// TwinCAT 3 PLC project Proj_Ueb_sw01
// ProgramVersion: 3.1.4023.0
// libraries:
//   Tc2_Standard, * (Beckhoff Automation GmbH)
//   Tc2_System, * (Beckhoff Automation GmbH)
//   Tc3_Module, * (Beckhoff Automation GmbH)
// project tree:
//   DUTs/ En_DistanceMode.TcDUT, En_ToggleMode.TcDUT
//   GVLs/ GVL_IO.TcGVL
//   / PlcTask.TcTTO
//   POUs/ Fb_MeanCalculatorWForgettingFactor.TcPOU, Fb_EdgeDetector.TcPOU, Fb_UltrasonicSensor.TcPOU, FUN_0to10V_TO_INT.TcPOU, FUN_Add.TcPOU, FUN_Divide.TcPOU, FUN_Multiply.TcPOU, FUN_Substract.TcPOU, MAIN.TcPOU, FUN_ShiftLeft.TcPOU, FUN_MeanCalculator.TcPOU, PRG_DoSomeMath.TcPOU
// (motion and I/O tree: see PLC project proj_sw01)
// real-time tasks:
//   TASK PlcTask: cycle T#10ms, priority 20, ADS port 350
//   TASK PlcTask1: cycle T#10ms, priority 21, ADS port 351
//   TASK PlcTask2: cycle T#10ms, priority 22, ADS port 352
// variable links:
//   Proj_Ueb_sw01/Proj_Ueb_sw01 Instance <-> Device 1 (EtherCAT)/Term 1 (EK1200)/Term 2 (EL1004)
//     PlcTask Inputs/GVL_IO.DI_BtnBlue <-> Channel 2/Input
//     PlcTask Inputs/GVL_IO.DI_BtnYellow <-> Channel 1/Input
//   Proj_Ueb_sw01/Proj_Ueb_sw01 Instance <-> Device 1 (EtherCAT)/Term 1 (EK1200)/Term 3 (EL2004)
//     PlcTask Outputs/GVL_IO.DO_LampGreen <-> Channel 2/Output
//     PlcTask Outputs/GVL_IO.DO_LampRed <-> Channel 1/Output
//   Proj_Ueb_sw01/Proj_Ueb_sw01 Instance <-> Device 1 (EtherCAT)/Term 1 (EK1200)/Term 4 (EL3004)
//     PlcTask Inputs/GVL_IO.AI_UltraSonicSensor <-> AI Standard Channel 1/Value
//   Proj_Ueb_sw01/Proj_Ueb_sw01 Instance <-> Device 1 (EtherCAT)/Term 1 (EK1200)/Term 5 (EL4034)
//     PlcTask Outputs/GVL_IO.AO_AnalogGauge <-> AO Outputs Channel 1/Analog output

CONFIGURATION Proj_Ueb_sw01
    RESOURCE PLC ON TwinCAT3
        TASK PlcTask(INTERVAL := T#10ms, PRIORITY := 21);
        PROGRAM MAIN WITH PlcTask : MAIN;
    END_RESOURCE
END_CONFIGURATION

// ---- DUTs/En_DistanceMode.TcDUT
{attribute 'qualified_only'}
{attribute 'strict'}
TYPE En_DistanceMode :
(
	Default := 0,
	NearerIsHigher,
	NearerIsLower
);
END_TYPE

// ---- DUTs/En_ToggleMode.TcDUT
{attribute 'qualified_only'}
{attribute 'strict'}
TYPE En_ToggleMode :
(
	Off := 0,
	Simulataneous,
	Alternating
);
END_TYPE

// ---- GVLs/GVL_IO.TcGVL
{attribute 'qualified_only'}
VAR_GLOBAL
	DI_BtnYellow 	AT %I* : BOOL;
	DI_BtnBlue	 	AT %I* : BOOL;
	
	DO_LampRed 		AT %Q* : BOOL;
	DO_LampGreen	AT %Q* : BOOL;
	
	AI_UltraSonicSensor  AT %I* : INT;
	AO_AnalogGauge		 AT %Q* : INT;
END_VAR

// ---- POUs/MAIN.TcPOU
PROGRAM MAIN
VAR
	f_Result 			:	REAL;
	i_Counter			: 	INT;
	f_RandomArray		: 	ARRAY[1..10] OF REAL := [5.0, 3.5, 4.6, 1.2, 13, 5.4, 5.6, 11.0, 15.6, 10];
	f_Product			: 	REAL;
	f_Sum 				: 	REAL;
	
	edgeDetectorBtnY	:   Fb_EdgeDetector;
	edgeDetectorBtnB	:   Fb_EdgeDetector;
	t_ToggleTime		: 	TIME := T#333MS;	// 1/Hz = [s]
	t_lastToggle		: 	TIME := TIME();
	togglingMode		: 	En_ToggleMode := En_ToggleMode.Off;
	b_LampR_On			: 	BOOL := FALSE;
	b_LampG_On			: 	BOOL := FALSE;
	
	ultraSonicSensorFb	:	Fb_UltrasonicSensor;
	
	a_lastValues		: 	ARRAY [1..NUM_STORED_VALS] OF REAL; 
	r_meanVal			: 	REAL := 0;
	fb_MeanCalc			: 	Fb_MeanCalculatorWForgettingFactor;
	r_forgettingFactor	: 	REAL := 0.5;
END_VAR
VAR CONSTANT
	NUM_STORED_VALS		: INT := 300;
END_VAR

// Aufgabe 1
f_Result := FUN_Add(1.3, 1.5);
f_Result := FUN_Add(3.3, 1000.5);
f_Result := FUN_Add(5.5, 51.5);

f_Result := FUN_Substract(1.3, 1);
f_Result := FUN_Substract(1.3, 2);

f_Result := FUN_Multiply(3, 1000);
f_Result := FUN_Multiply(55, 5.55);

f_Result := FUN_Divide(9, 3);
f_Result := FUN_Divide(55, 0);


// Aufgabe 3
// Call program
PRG_DoSomeMath.f_Inp1 := 1.5;
PRG_DoSomeMath.f_Inp2 := 5.4;
PRG_DoSomeMath();
// Access program variables
f_Result := PRG_DoSomeMath.f_AddResult;
i_Counter := PRG_DoSomeMath.i_CallCounter;


// Aufgabe 7 & 8
// insert first values
f_Product := f_RandomArray[1];
f_Sum := f_RandomArray[1];
// for loop
FOR i_Counter := 2 TO 10 DO
	f_Product 	:= f_Product * f_RandomArray[i_Counter];
	f_Sum		:= f_Sum + f_RandomArray[i_Counter];
END_FOR

// Aufgabe 9
// insert first values
f_Product := f_RandomArray[1];
f_Sum := f_RandomArray[1];
i_Counter := 2;
// while loop
WHILE i_Counter <= 10 DO
	f_Product 	:= f_Product * f_RandomArray[i_Counter];
	f_Sum		:= f_Sum + f_RandomArray[i_Counter];
	i_Counter 	:= i_Counter + 1;
END_WHILE

// Aufgabe 10
// insert first values
f_Product := f_RandomArray[1];
f_Sum := f_RandomArray[1];
i_Counter := 2;
// do while loop = repeat loop
REPEAT
	f_Product 	:= f_Product * f_RandomArray[i_Counter];
	f_Sum		:= f_Sum + f_RandomArray[i_Counter];
	i_Counter 	:= i_Counter + 1;
UNTIL i_Counter > 10
END_REPEAT


// Aufgabe 11 and 12
edgeDetectorBtnY(inputValue := GVL_IO.DI_BtnYellow);
edgeDetectorBtnB(inputValue := GVL_IO.DI_BtnBlue);

// double press?
IF edgeDetectorBtnB.doublePress OR edgeDetectorBtnY.doublePress THEN
	t_ToggleTime := t_ToggleTime / 2;  // double frequency
END_IF

// triple press?
IF edgeDetectorBtnB.triplePress OR edgeDetectorBtnY.triplePress THEN
	t_ToggleTime := t_ToggleTime * 2;  // half frequency
END_IF

CASE togglingMode OF
	
	/// CASE OFF ///
	En_ToggleMode.Off:
	// lamp actions
	b_LampR_On := FALSE;
	b_LampG_On := FALSE;
	t_ToggleTime := T#333MS; // reset to default time
	
	// switch mode
	IF edgeDetectorBtnY.risingEdge THEN
		togglingMode := En_ToggleMode.Simulataneous;
	END_IF
	IF edgeDetectorBtnB.risingEdge THEN 
		togglingMode := En_ToggleMode.Alternating;
		b_LampG_On := TRUE;  // initial lamp on => alternating
	END_IF
	
	/// CASE Simulataneous ///
	En_ToggleMode.Simulataneous:
	// lamp actions
	IF((t_lastToggle + t_ToggleTime) < TIME()) THEN
		b_LampR_On := NOT b_LampR_On;
		b_LampG_On := NOT b_LampG_On;
		t_lastToggle := TIME();
	END_IF
	
	// switch mode
	IF edgeDetectorBtnY.risingEdge THEN
		togglingMode := En_ToggleMode.Off;
	END_IF
	

	/// CASE ALTERNATING ///
	En_ToggleMode.Alternating:
	// lamp actions
	IF((t_lastToggle + t_ToggleTime) < TIME()) THEN
		b_LampR_On := NOT b_LampR_On;
		b_LampG_On := NOT b_LampG_On;
		t_lastToggle := TIME();
	END_IF
	
	// switch mode
	IF edgeDetectorBtnB.risingEdge THEN
		togglingMode := En_ToggleMode.Off;
	END_IF

	
END_CASE


GVL_IO.DO_LampRed := b_LampR_On;
GVL_IO.DO_LampGreen := b_LampG_On;


// Aufgabe 13
ultraSonicSensorFb(	i_UltraSonicAnalogInput := GVL_IO.AI_UltraSonicSensor, 
					e_DistanceMode := En_DistanceMode.NearerIsHigher);
GVL_IO.AO_AnalogGauge := ultraSonicSensorFb.i_AnalogOutput;

// Aufgabe 14
FUN_ShiftLeft(a_Values := a_lastValues);  // shift array left
a_lastValues[NUM_STORED_VALS] := ultraSonicSensorFb.r_VoltageUltraSonicSensor;  // store last value

// Aufgabe 15
fb_MeanCalc(r_inputValue := ultraSonicSensorFb.r_VoltageUltraSonicSensor, r_forgettingFactor := r_forgettingFactor);
r_meanVal := fb_MeanCalc.r_meanValueOutput;
GVL_IO.AO_AnalogGauge := FUN_0to10V_TO_INT(r_AnalogValue0to10V := r_meanVal);

END_PROGRAM

// ---- POUs/Fb_EdgeDetector.TcPOU
FUNCTION_BLOCK INTERNAL Fb_EdgeDetector
VAR_INPUT
	inputValue		: BOOL;
END_VAR
VAR_OUTPUT
	risingEdge		: BOOL;
	fallingEdge		: BOOL;
	doublePress		: BOOL;
	triplePress		: BOOL;
END_VAR
VAR
	i_risingEdgCnt			: INT := 0;  		// internal var
	lastValue 				: BOOL;				// last value registered
	tlastPush				: TIME := TIME();	// time when last push happened
	tLastRising				: TIME := TIME();	// time when last rising edge happened
	tDebounce	    		: TIME := T#20MS;   // time to debounce input value
	tMultiPressTime			: TIME := T#200MS;	// time between which multiple presses to allow the user to press button again
	
END_VAR

// reset output signals
fallingEdge := FALSE;
risingEdge := FALSE;
doublePress := FALSE;
triplePress := FALSE;

// if a change happened and new values get accepted
IF(inputValue <> lastValue AND (tlastPush + tDebounce) < TIME()) THEN
	IF(inputValue) THEN
		i_risingEdgCnt := i_risingEdgCnt + 1;
		
		tLastRising := TIME(); // reset last rising time (give another tMultiPressTime time to press the button another time
	ELSE
		fallingEdge := TRUE;
	END_IF
	lastValue := inputValue;  // overwrite stored value
	tlastPush := TIME();
END_IF


// handle rising edge (with double press)
CASE i_risingEdgCnt OF
	1:
	IF (tLastRising + tMultiPressTime) < TIME() THEN
		risingEdge := TRUE;
		i_risingEdgCnt := 0;
	END_IF
	
	2:
	IF (tLastRising + tMultiPressTime) < TIME() THEN
		doublePress := TRUE;
		i_risingEdgCnt := 0;
	END_IF
	
	3:
	// instantly report triple press, since no more amount of multi press is output
	triplePress := TRUE;
	i_risingEdgCnt := 0;
ELSE
	;
END_CASE

END_FUNCTION_BLOCK

// ---- POUs/Fb_UltrasonicSensor.TcPOU
FUNCTION_BLOCK Fb_UltrasonicSensor
VAR_INPUT
	i_UltraSonicAnalogInput		: INT;
	e_DistanceMode				: En_DistanceMode := En_DistanceMode.Default;
END_VAR
VAR_OUTPUT
	r_VoltageUltraSonicSensor	: REAL;
	i_AnalogOutput				: INT;
END_VAR
VAR
	l_UltraSonic				: DINT;
END_VAR
VAR CONSTANT
	MAX_VOLTAGE					: REAL := 10.0;
	MAX_INT						: INT := 32767;
END_VAR

// multiply by max voltage
l_UltraSonic := i_UltraSonicAnalogInput * REAL_TO_INT(MAX_VOLTAGE);

// divide by resolution
r_VoltageUltraSonicSensor := DINT_TO_REAL(l_UltraSonic) / INT_TO_REAL(MAX_INT);

// check distance mode and calculate
IF(e_DistanceMode = En_DistanceMode.NearerIsHigher) THEN
	l_UltraSonic := MAX_INT - i_UltraSonicAnalogInput;
ELSE
	l_UltraSonic := i_UltraSonicAnalogInput;
END_IF

// analog output, dint wont be larger than int at this point
i_AnalogOutput := DINT_TO_INT(l_UltraSonic);

END_FUNCTION_BLOCK

// ---- POUs/Fb_MeanCalculatorWForgettingFactor.TcPOU
FUNCTION_BLOCK Fb_MeanCalculatorWForgettingFactor
VAR_IN_OUT
	r_inputValue			: REAL;
	r_forgettingFactor		: REAL;
END_VAR
VAR_OUTPUT
	r_meanValueOutput		: REAL;
END_VAR
VAR
	r_meanValue				: REAL;
	lr_numerator			: LREAL;
	lr_denominator			: LREAL;
	lr_forgFactorExp		: LREAL;
	i_counter				: DINT;
END_VAR

r_meanValue := (r_forgettingFactor * r_meanValue) + (1-r_forgettingFactor) * r_inputValue;
r_meanValueOutput := r_meanValue;

END_FUNCTION_BLOCK

// ---- POUs/FUN_Add.TcPOU
FUNCTION FUN_Add : REAL
VAR_INPUT
		f_Inp1			: REAL;
		f_Inp2			: REAL;
END_VAR
VAR
END_VAR

FUN_Add := f_Inp1 + f_Inp2;

END_FUNCTION

// ---- POUs/FUN_Substract.TcPOU
FUNCTION FUN_Substract : REAL
VAR_INPUT
		f_Inp1			: REAL;
		f_Inp2			: REAL;
END_VAR
VAR
END_VAR

FUN_Substract := f_Inp1 - f_Inp2;

END_FUNCTION

// ---- POUs/FUN_Multiply.TcPOU
FUNCTION FUN_Multiply : REAL
VAR_INPUT
		f_Inp1			: REAL;
		f_Inp2			: REAL;
END_VAR
VAR
END_VAR

FUN_Multiply := f_Inp1 * f_Inp2;

END_FUNCTION

// ---- POUs/FUN_Divide.TcPOU
FUNCTION FUN_Divide : REAL
VAR_INPUT
		f_Inp1			: REAL;
		f_Inp2			: REAL;
END_VAR
VAR
END_VAR

IF(f_Inp2 = 0) THEN
	FUN_Divide := 0;
ELSE
	FUN_Divide := f_Inp1 / f_Inp2;
END_IF

END_FUNCTION

// ---- POUs/PRG_DoSomeMath.TcPOU
PROGRAM PRG_DoSomeMath
VAR_INPUT
	f_Inp1				: REAL;
	f_Inp2				: REAL;
END_VAR
VAR
	f_AddResult 		: REAL;
	f_SubstractResult 	: REAL;
	f_MultiplyResult 	: REAL;
	f_DivideResult 		: REAL;
	i_CallCounter		: INT;
END_VAR

// Increment call counter
i_CallCounter := i_CallCounter + 1;

f_AddResult 		:= FUN_Add(f_Inp1, f_Inp2);
f_SubstractResult 	:= FUN_Substract(f_Inp1, f_Inp2);
f_MultiplyResult 	:= FUN_Multiply(f_Inp1, f_Inp2);
f_DivideResult 		:= FUN_Divide(f_Inp1, f_Inp2);

END_PROGRAM

// ---- POUs/FUN_ShiftLeft.TcPOU
FUNCTION FUN_ShiftLeft : BOOL
VAR_IN_OUT
	a_Values	: ARRAY [*] OF REAL;
END_VAR
VAR
	i_counter	: DINT := 0;
END_VAR

FOR i_counter:=LOWER_BOUND(a_Values,1) TO UPPER_BOUND(a_Values,1) DO
	a_Values[i_counter] := a_Values[i_counter + 1];
END_FOR;

END_FUNCTION

// ---- POUs/FUN_0to10V_TO_INT.TcPOU
FUNCTION FUN_0to10V_TO_INT : INT
VAR_INPUT
	r_AnalogValue0to10V		: REAL;
END_VAR
VAR
	i_Val					: DINT;
END_VAR
VAR CONSTANT
	MAX_VOLTAGE				: REAL := 10.0;
	MAX_INT					: INT := 32767;
END_VAR

// Multiply
i_Val := REAL_TO_DINT(r_AnalogValue0to10V * INT_TO_REAL(MAX_INT));

// divide by 10, convert to int
FUN_0to10V_TO_INT := DINT_TO_INT(i_Val / REAL_TO_INT(MAX_VOLTAGE));

END_FUNCTION

// ---- POUs/FUN_MeanCalculator.TcPOU
FUNCTION FUN_MeanCalculator : REAL
VAR_IN_OUT
	a_Values	: ARRAY [*] OF REAL;
END_VAR
VAR
	i_counter	: DINT;
	lr_MeanVal	: LREAL;
END_VAR

// reset
lr_MeanVal := 0;

FOR i_counter:=LOWER_BOUND(a_Values,1) TO UPPER_BOUND(a_Values,1) DO
	lr_MeanVal := lr_MeanVal + a_Values[i_counter];
END_FOR;

FUN_MeanCalculator := lr_MeanVal / UPPER_BOUND(a_Values,1);

END_FUNCTION
